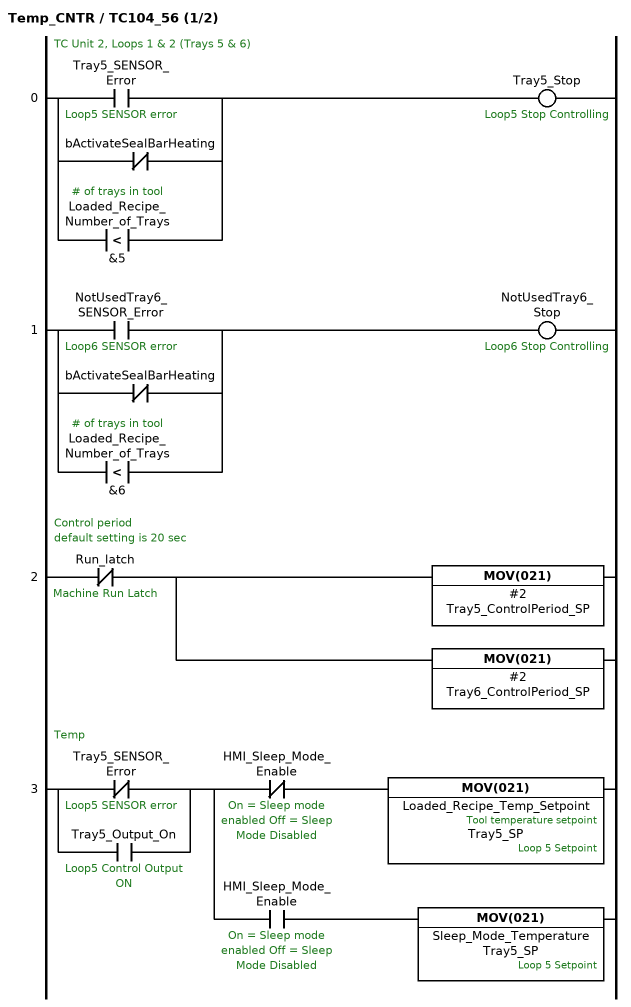
; [picture p168: Temp_CNTR / TC104_56, rungs 0-3]
; rung 0: TC Unit 2, Loops 1 & 2 (Trays 5 & 6)
LD Tray5_SENSOR_Error  ; Loop5 SENSOR error
ORNOT bActivateSealBarHeating
OR<(310) Loaded_Recipe_Number_of_Trays &5  ; # of trays in tool
OUT Tray5_Stop  ; Loop5 Stop Controlling
; rung 1
LD NotUsedTray6_SENSOR_Error  ; Loop6 SENSOR error
ORNOT bActivateSealBarHeating
OR<(310) Loaded_Recipe_Number_of_Trays &6  ; # of trays in tool
OUT NotUsedTray6_Stop  ; Loop6 Stop Controlling
; rung 2: Control period / default setting is 20 sec
LDNOT Run_latch  ; Machine Run Latch
MOV(021) #2 Tray5_ControlPeriod_SP
MOV(021) #2 Tray6_ControlPeriod_SP
; rung 3: Temp
LDNOT Tray5_SENSOR_Error  ; Loop5 SENSOR error
OR Tray5_Output_On  ; Loop5 Control Output ON
OUT TR0
ANDNOT HMI_Sleep_Mode_Enable  ; On = Sleep mode enabled Off = Sleep Mode Disabled
MOV(021) Loaded_Recipe_Temp_Setpoint Tray5_SP  ; Tool temperature setpoint, Loop 5 Setpoint
LD TR0
AND HMI_Sleep_Mode_Enable  ; On = Sleep mode enabled Off = Sleep Mode Disabled
MOV(021) Sleep_Mode_Temperature Tray5_SP  ; Loop 5 Setpoint

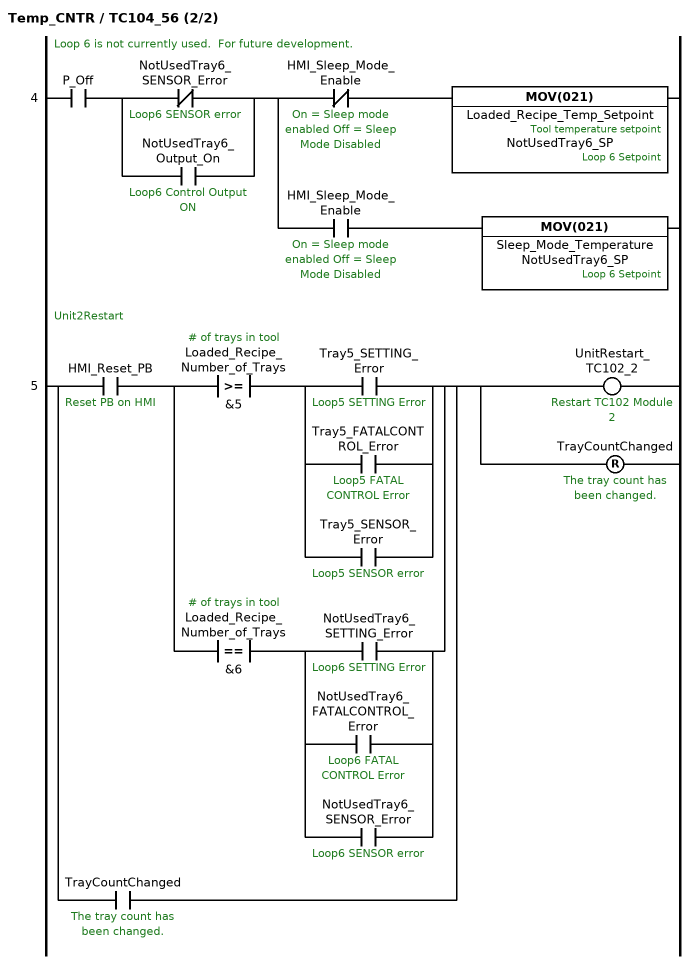
; rung 4: Loop 6 is not currently used.  For future development.
LD P_Off
LDNOT NotUsedTray6_SENSOR_Error  ; Loop6 SENSOR error
OR NotUsedTray6_Output_On  ; Loop6 Control Output ON
ANDLD
OUT TR0
ANDNOT HMI_Sleep_Mode_Enable  ; On = Sleep mode enabled Off = Sleep Mode Disabled
MOV(021) Loaded_Recipe_Temp_Setpoint NotUsedTray6_SP  ; Tool temperature setpoint, Loop 6 Setpoint
LD TR0
AND HMI_Sleep_Mode_Enable  ; On = Sleep mode enabled Off = Sleep Mode Disabled
MOV(021) Sleep_Mode_Temperature NotUsedTray6_SP  ; Loop 6 Setpoint
; rung 5: Unit2Restart
LD HMI_Reset_PB  ; Reset PB on HMI
LD>=(325) Loaded_Recipe_Number_of_Trays &5  ; # of trays in tool
LD Tray5_SETTING_Error  ; Loop5 SETTING Error
OR Tray5_FATALCONTROL_Error  ; Loop5 FATAL CONTROL Error
OR Tray5_SENSOR_Error  ; Loop5 SENSOR error
ANDLD
LD=(300) Loaded_Recipe_Number_of_Trays &6  ; # of trays in tool
LD NotUsedTray6_SETTING_Error  ; Loop6 SETTING Error
OR NotUsedTray6_FATALCONTROL_Error  ; Loop6 FATAL CONTROL Error
OR NotUsedTray6_SENSOR_Error  ; Loop6 SENSOR error
ANDLD
ORLD
ANDLD
OR TrayCountChanged  ; The tray count has been changed.
OUT UnitRestart_TC102_2  ; Restart TC102 Module 2
RSET TrayCountChanged  ; The tray count has been changed.

### Section END
; rung 0
END(001)

## Function block Average
VAR_INPUT
  Height_memory1 : INT;
  Height_memory2 : INT;
  Height_memory3 : INT;
  Height_memory4 : INT;
  Height_memory5 : INT;
  Number_of_Trays : INT;
END_VAR
VAR_OUTPUT
  Average_height : INT;
END_VAR
VAR
  calculation : REAL;
  Total : INT;
  converted_total : REAL;
END_VAR
Total:= Height_memory1+Height_memory2+Height_memory3+Height_memory4+Height_memory5;

converted_total:= INT_TO_REAL(Total);

calculation:= converted_total/INT_TO_REAL(Number_of_Trays);

Average_height:= REAL_TO_INT(calculation);

## Function block C_to_F
VAR_INPUT
  Celcius : INT;
END_VAR
VAR_OUTPUT
  F : INT;
END_VAR
F:= REAL_TO_INT(INT_TO_REAL(Celcius)*9.0/5.0+320.0);

## Function block Conv_Scale_analog_with_Int_range
VAR_INPUT
  Analog_input : INT;
  Zero_point : REAL;  (* This is the scaled value when the analog input is 0. *)
  Max_Point : REAL;  (* This is the scaled value for the maximum analog input 8000 in this example (4000 if set to 4000 in the I/O Table). *)
  Max_Analog_In_INT : INT;  (* The maximum value of your analog input.  For instance, if the analog input range is 0-8000, enter &8000 as the input to the block. *)
END_VAR
VAR_OUTPUT
  Scaled_Real_output : REAL;
  Scaled_Integer_Output : INT;
  Scaled_BCD_Output : WORD;
END_VAR
VAR
  Input_real : REAL;
  Slope : REAL;
  Intercept : REAL;
END_VAR
Input_real:=INT_TO_REAL(Analog_input);

Slope:= (Max_Point-Zero_point)/int_to_real(Max_Analog_In_INT);
Intercept:= Max_Point-Slope*int_to_real(Max_Analog_In_INT);
	
Scaled_Real_output:= Slope*Input_real+Intercept;
Scaled_Integer_Output:= REAL_TO_INT(Scaled_Real_output);
Scaled_BCD_Output:= INT_TO_BCD_WORD(Scaled_Integer_Output);

## Function block F_to_C
VAR_INPUT
  F : INT;
END_VAR
VAR_OUTPUT
  Celcius : INT;
END_VAR
Celcius:= REAL_TO_INT((INT_TO_REAL(F)-320.0)*5.0/9.0);

## Function block Film_Scaling
VAR
  Accel_Pulses_s_4ms_Real : REAL;
  Decel_Pulses_s_4ms_Real : REAL;
  Film_Dist_Pulses_Real : REAL;
  Film_Velocity_Pulses_Real : REAL;
  Roll_Circ_mm : REAL := 159.5929;  (* $?St$Bk?_#[14] / 2" diameter roll x pi x 25.4$?St$Bk?_#[14] *)
END_VAR
Overall_ratio:= Gear_Ratio*Pulses_Rev/Roll_Circ_mm;
Film_Velocity_Pulses_Real:= INT_TO_REAL(Velocity)*Overall_ratio;
Film_Velocity_Pulses:= REAL_TO_DINT(Film_Velocity_Pulses_Real);
Accel_Pulses_s_4ms_Real:= INT_TO_REAL(Accel)*Overall_ratio/+250.0;
Accel_Pulses_s_4ms:= REAL_TO_INT(Accel_Pulses_s_4ms_Real);
Decel_Pulses_s_4ms_Real:= INT_TO_REAL(Decel)*Overall_ratio/+250.0;
Decel_Pulses_s_4ms:= REAL_TO_INT(Decel_Pulses_s_4ms_Real);
Film_Dist_Pulses_Real:= INT_TO_REAL(Film_Feed_Dist)*Overall_ratio;
Film_Dist_Pulses:= REAL_TO_DINT(Film_Dist_Pulses_Real);
Film_Dist_Pulses_Real:= INT_TO_REAL(Registration_distance)*Overall_ratio;
Film_Dist_Reg:= REAL_TO_DINT(Film_Dist_Pulses_Real);
Yank_Dist_Pulses_Real:= INT_TO_REAL(Yank_Dist)*Overall_ratio;
Yank_Dist_Pulses:= REAL_TO_DINT(Yank_Dist_Pulses_Real);
Yank_Dist_Neg:= Yank_Dist_Pulses*-1;
Slow_Down_Speed_Real:= INT_TO_REAL(Slow_Down_Speed)*Overall_ratio;
Slow_Down_Speed_Out:= REAL_TO_DINT(Slow_Down_Speed_Real);
Film_Dist_Slow_Pulses_Real:= INT_TO_REAL(Slow_Down_Distance)*Overall_ratio;
Film_Dist_Slow_Pulses:= REAL_TO_DINT(Film_Dist_Slow_Pulses_Real);

## Function block Minimum_Distance_Calc
VAR_INPUT
  Velocity : DINT;
  Decel_Setting : INT;
END_VAR
VAR_OUTPUT
  Minimum_Distance : DINT;
END_VAR
VAR
  Velocity_Real : REAL;
  Decel_Real : REAL;
  CalcA : REAL;  (* Calc A from help file *)
  Time_to_Decel : REAL;
  CalcB : REAL;  (* Calculation B from help file *)
END_VAR
Velocity_Real:= DINT_TO_REAL(Velocity);
Decel_Real:= INT_TO_REAL(Decel_Setting);
Time_to_Decel:= Velocity_Real/(Decel_Real/0.004);
CalcA:= Velocity_Real*Time_to_Decel/2.0+0.5;
CalcB:= Velocity_Real*0.004+0.5;
Minimum_Distance:= REAL_TO_DINT(CalcA)+REAL_TO_DINT(CalcB)*4;

## Function block offsetC_to_offsetF
; This function block takes an offset in celcius and converts it to an offset in Fahrenheit
VAR_INPUT
  Celcius_Offset : INT;
END_VAR
VAR_OUTPUT
  Fahrenheit_Offset : INT;
END_VAR
Fahrenheit_Offset:= REAL_TO_INT((+9.0/+5.0)*INT_TO_REAL(Celcius_Offset));

## Function block OffsetF_to_OffsetC
; Converts an offset from F to C.
VAR_INPUT
  Fahr_Offset : INT;
END_VAR
VAR_OUTPUT
  Celcius_Offset : INT;
END_VAR
Celcius_Offset:= REAL_TO_INT((+5.0/+9.0)*INT_TO_REAL(Fahr_Offset));

## Function block Scale_Gas_range
VAR_INPUT
  Analog_input : INT;
  Zero_point : REAL;  (* This is the scaled value when the analog input is 0. *)
  Max_Point : REAL;  (* This is the scaled value for the maximum analog input 8000 in this example (4000 if set to 4000 in the I/O Table). *)
  Max_Analog_In_INT : INT;  (* The maximum value of your analog input.  For instance, if the analog input range is 0-8000, enter &8000 as the input to the block. *)
END_VAR
VAR_OUTPUT
  Scaled_Real_output : REAL;
  Scaled_Integer_Output : INT;
  Scaled_BCD_Output : WORD;
END_VAR
VAR
  Input_real : REAL;
  Slope : REAL;
  Intercept : REAL;
END_VAR
Input_real:=INT_TO_REAL(Analog_input);

Slope:= (Max_Point-Zero_point)/int_to_real(Max_Analog_In_INT);
Intercept:= Max_Point-Slope*int_to_real(Max_Analog_In_INT);
	
Scaled_Real_output:= Slope*Input_real+Intercept;
Scaled_Integer_Output:= REAL_TO_INT(Scaled_Real_output);
Scaled_BCD_Output:= INT_TO_BCD_WORD(Scaled_Integer_Output);

## Function block TPM_Calc
VAR_INPUT
  Cycle_Time : UINT;  (* Cycle time in 1/100s of a second *)
  Num_of_Trays : INT;
END_VAR
VAR_OUTPUT
  TPM : UINT;  (* Trays per minute in 1/10 of a TPM *)
END_VAR
VAR
  Cycle_Time_real : REAL;
  TPM_Real : REAL;
END_VAR
Cycle_Time_real:= UINT_TO_REAL(Cycle_Time)/100.0;
TPM_Real:= 60.0/Cycle_Time_real*INT_TO_REAL(Num_of_Trays);
TPM:= REAL_TO_UINT(TPM_Real*10.0);

## Function block Vac_Test_Calc
VAR_INPUT
  Leak_Pressure : UINT;
  Target_Pressure : UINT;
  Leak_Time : UINT;
END_VAR
VAR_OUTPUT
  Leak_Rate : UINT;  (* In tenths of an Mbar per second *)
END_VAR
VAR
  Leak_Pressure_Real : REAL;
  Target_Pressure_Real : REAL;
  Leak_Time_Real : REAL;
  Leak_Rate_Real : REAL;
END_VAR
Target_Pressure_Real:= UINT_TO_REAL(Target_Pressure);
Leak_Pressure_Real:= UINT_TO_REAL(Leak_Pressure);
Leak_Time_Real:= UINT_TO_REAL(Leak_Time)/100.0;
Leak_Rate_Real:=(Leak_Pressure_Real-Target_Pressure_Real)/Leak_Time_Real;
Leak_Rate:= REAL_TO_UINT(Leak_Rate_Real*10.0);

## Function block Vel_ACC_DEC_Scale
VAR_INPUT
  Vel_Percent : UINT;
  Acc_Percent : UINT;
  Dec_Percent : UINT;
END_VAR
VAR_OUTPUT
  Vel_Scaled : UDINT;
  ACC_Scaled : UINT;
  DEC_Scaled : UINT;
END_VAR
VAR
  Real_Vel_Percent : REAL;
  Real_ACC_Percent : REAL;
  Real_DEC_Percent : REAL;
  Real_Vel_Scaled : REAL;
  Real_ACC_Scaled : REAL;
  Real_DEC_Scaled : REAL;
END_VAR
(*Convert all inputs to real numbers*)
Real_Vel_Percent:= UINT_TO_REAL(Vel_Percent);
Real_ACC_Percent:= UINT_TO_REAL(Acc_Percent);
Real_DEC_Percent:= UINT_TO_REAL(Dec_Percent);
(*Scale the converted values  
1000.0 is the 0% value for speed, ACC and DEC
26500 is the 100% for velocity and
99999 is the 100% value for ACC and DEC *)
Real_Vel_Scaled:= (26500.0-1000.0)*Real_Vel_Percent/100.0+1000.0;
Real_ACC_Scaled:= ((99999.0-1000.0)*Real_ACC_Percent/100.0+1000.0)/250.0;
Real_DEC_Scaled:= ((99999.0-1000.0)*Real_DEC_Percent/100.0+1000.0)/250.0;
(*Convert answers back to UDINT for output*)
Vel_Scaled:= REAL_TO_UDINT(Real_Vel_Scaled);
ACC_Scaled:= REAL_TO_UINT(Real_ACC_Scaled);
DEC_Scaled:= REAL_TO_UINT(Real_DEC_Scaled);